PROGRAM Servo
VAR
	fbServoVise				: FB_ServoVise;
END_VAR

fbVisePos();
fbServoVise(
	bErrorAck:= , 
	bEnable:= , 
	eCommand:= , 
	bManualMode:= , 
	lrTargetDistance:= , 
	lrVisePosition:= fbVisePos.nDistance, 
	bVisePosValid:= fbVisePos.bValid, 
	nTargetVelocity:= , 
	nTorque:= , 
	nTorqueRamp:= , 
	nTorqueVelocityLimit:= , 
	nOverride:= , 
	nAttachDistance:= , 
	nAttachVelocity:= , 
	stAxisEvent:= , 
	bReady=> , 
	bBusy=> , 
	bDone=> , 
	bError=> );

END_PROGRAM

(* stored: Version 1.1.0.1, ProductVersion 3.1.4024.12
   POU Servo: Id {7c80c4b6-5bdf-4d78-8a31-a44be7b9eb1b}, SpecialFunc None *)
